FUNCTION_BLOCK AX_AND_3 (* FB to calculate boolean AND *)
  (* Standard: 61499-2; Description: Copyright (c) 2024 HR Agrartechnik GmbH This program and the accompanying materials are made available under the terms of the Eclipse Public License 2.0 which is available at https://www.eclipse.org/legal/epl-2.0/ SPDX-License-Identifier: EPL-2.0 *)
  (* Version 1.0, 2024-10-23, Franz Höpfinger, HR Agrartechnik GmbH *)
  {SET_ATTRIBUTE(eclipse4diac::core::GenericClassName, 'GEN_AX_AND')}
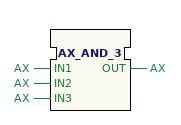
  SOCKETS
    IN1 : AX; (* AND input 1 *)
    IN2 : AX; (* AND input 2 *)
    IN3 : AX; (* AND input 3 *)
  END_SOCKETS
  PLUGS
    OUT : AX; (* AND result *)
  END_PLUGS
END_FUNCTION_BLOCK
